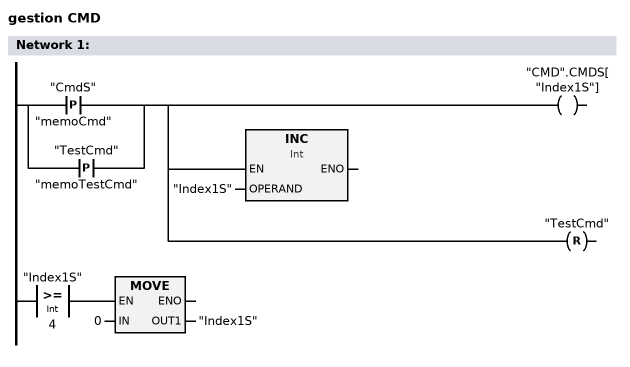
   RUNG wire#powerrail
      P_Contact(operand := "CmdS", bit := "memoCmd")
      wire#w1
      Coil( "CMD".CMDS["Index1S"] )
   END_RUNG
   RUNG wire#powerrail
      P_Contact(operand := "TestCmd", bit := "memoTestCmd")
   END_RUNG wire#w1
   RUNG wire#w1
      { S7_Templates := "DestType := Int" } Inc( "Index1S" )
   END_RUNG
   RUNG wire#w1
      R_Coil( "TestCmd" )
   END_RUNG
   RUNG wire#powerrail
      { S7_Templates := "SrcType := Int" } GE_Contact(in1 := "Index1S", in2 := 4)
      Move(in := 0, out1 => "Index1S")
   END_RUNG
   // the same network as SCL:
   #_w1 := "CmdS" AND NOT "memoCmd";   // rising edge of "CmdS"
   "memoCmd" := "CmdS";
   #_w2 := "TestCmd" AND NOT "memoTestCmd";   // rising edge of "TestCmd"
   "memoTestCmd" := "TestCmd";
   "CMD".CMDS["Index1S"] := #_w1 OR #_w2;
   IF #_w1 OR #_w2 THEN
       "Index1S" := "Index1S" + 1;
       "TestCmd" := FALSE;
   END_IF;
   IF "Index1S" >= 4 THEN "Index1S" := 0; END_IF;
END_REGION

REGION Network 2 (SCL)
   IF "TestX40" AND NOT "CMD".CMDFinal_S THEN
       IF "CMD".CMDS["index2S"] = TRUE THEN
           "CMD".CMDFinal_S := TRUE;
           "CMD".CMDS["index2S"] := 0;
       ELSE
           "index2S" := "index2S" + 1;
           IF "index2S" >= 4 THEN
               "index2S" := 0;
           END_IF;
       END_IF;
   END_IF;
END_REGION
END_FUNCTION

ORGANIZATION_BLOCK "Main"   // OB1, LAD, ProgramCycle
{ S7_Optimized_Access := 'TRUE' }
VERSION : 0.1
   VAR_INPUT
      Initial_Call : Bool;
      Remanence : Bool;
   END_VAR
BEGIN

REGION Network 1
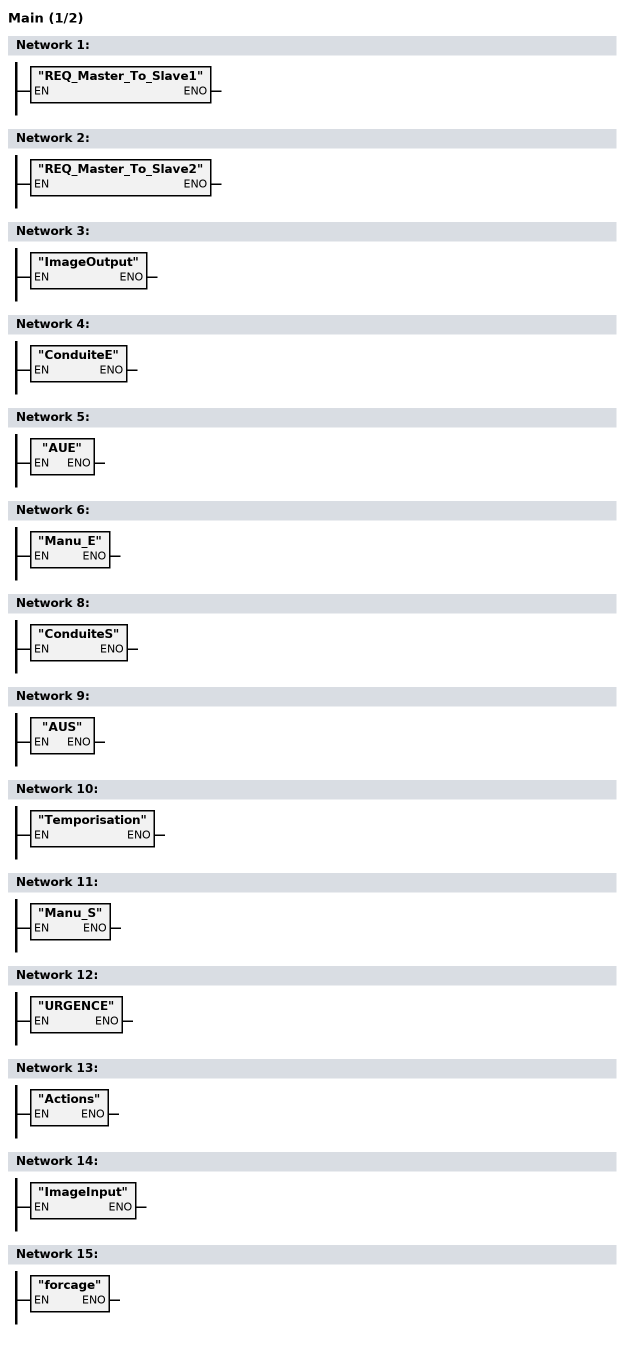
   RUNG wire#powerrail
      "REQ_Master_To_Slave1"()
   END_RUNG
   // the same network as SCL:
   "REQ_Master_To_Slave1"();
END_REGION

REGION Network 2
   RUNG wire#powerrail
      "REQ_Master_To_Slave2"()
   END_RUNG
   // the same network as SCL:
   "REQ_Master_To_Slave2"();
END_REGION

REGION Network 3
   RUNG wire#powerrail
      "ImageOutput"()
   END_RUNG
   // the same network as SCL:
   "ImageOutput"();
END_REGION

REGION Network 4
   RUNG wire#powerrail
      "ConduiteE"()
   END_RUNG
   // the same network as SCL:
   "ConduiteE"();
END_REGION

REGION Network 5
   RUNG wire#powerrail
      "AUE"()
   END_RUNG
   // the same network as SCL:
   "AUE"();
END_REGION

REGION Network 6
   RUNG wire#powerrail
      "Manu_E"()
   END_RUNG
   // the same network as SCL:
   "Manu_E"();
END_REGION

REGION Network 8
   RUNG wire#powerrail
      "ConduiteS"()
   END_RUNG
   // the same network as SCL:
   "ConduiteS"();
END_REGION

REGION Network 9
   RUNG wire#powerrail
      "AUS"()
   END_RUNG
   // the same network as SCL:
   "AUS"();
END_REGION

REGION Network 10
   RUNG wire#powerrail
      "Temporisation"()
   END_RUNG
   // the same network as SCL:
   "Temporisation"();
END_REGION

REGION Network 11
   RUNG wire#powerrail
      "Manu_S"()
   END_RUNG
   // the same network as SCL:
   "Manu_S"();
END_REGION

REGION Network 12
   RUNG wire#powerrail
      "URGENCE"()
   END_RUNG
   // the same network as SCL:
   "URGENCE"();
END_REGION

REGION Network 13
   RUNG wire#powerrail
      "Actions"()
   END_RUNG
   // the same network as SCL:
   "Actions"();
END_REGION

REGION Network 14
   RUNG wire#powerrail
      "ImageInput"()
   END_RUNG
   // the same network as SCL:
   "ImageInput"();
END_REGION

REGION Network 15
   RUNG wire#powerrail
      "forcage"()
   END_RUNG
   // the same network as SCL:
   "forcage"();
END_REGION

REGION Network 16
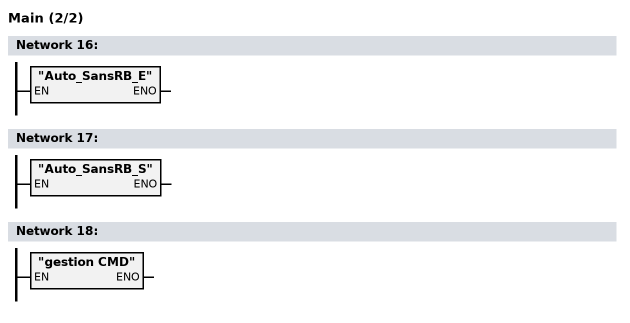
   RUNG wire#powerrail
      "Auto_SansRB_E"()
   END_RUNG
   // the same network as SCL:
   "Auto_SansRB_E"();
END_REGION

REGION Network 17
   RUNG wire#powerrail
      "Auto_SansRB_S"()
   END_RUNG
   // the same network as SCL:
   "Auto_SansRB_S"();
END_REGION

REGION Network 18
   RUNG wire#powerrail
      "gestion CMD"()
   END_RUNG
   // the same network as SCL:
   "gestion CMD"();
END_REGION
END_ORGANIZATION_BLOCK

ORGANIZATION_BLOCK "Startup"   // OB100, LAD, Startup
TITLE = "Complete Restart"
{ S7_Optimized_Access := 'TRUE' }
VERSION : 0.1
   VAR_INPUT
      LostRetentive : Bool;   // True if retentive data are lost
      LostRTC : Bool;   // True if date and time are lost
   END_VAR
BEGIN

REGION Network 1
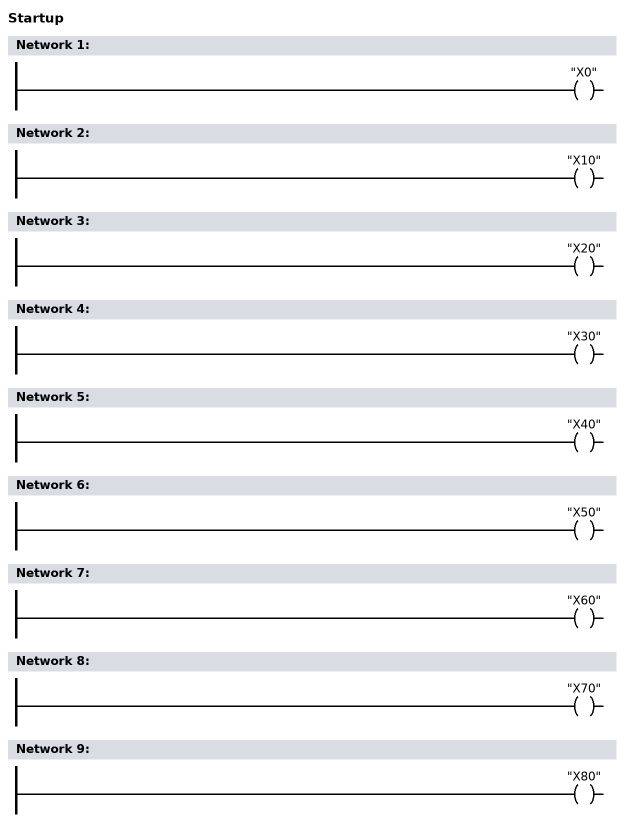
   RUNG wire#powerrail
      Coil( "X0" )
   END_RUNG
   // the same network as SCL:
   "X0" := TRUE;
END_REGION

REGION Network 2
   RUNG wire#powerrail
      Coil( "X10" )
   END_RUNG
   // the same network as SCL:
   "X10" := TRUE;
END_REGION

REGION Network 3
   RUNG wire#powerrail
      Coil( "X20" )
   END_RUNG
   // the same network as SCL:
   "X20" := TRUE;
END_REGION

REGION Network 4
   RUNG wire#powerrail
      Coil( "X30" )
   END_RUNG
   // the same network as SCL:
   "X30" := TRUE;
END_REGION

REGION Network 5
   RUNG wire#powerrail
      Coil( "X40" )
   END_RUNG
   // the same network as SCL:
   "X40" := TRUE;
END_REGION

REGION Network 6
   RUNG wire#powerrail
      Coil( "X50" )
   END_RUNG
   // the same network as SCL:
   "X50" := TRUE;
END_REGION

REGION Network 7
   RUNG wire#powerrail
      Coil( "X60" )
   END_RUNG
   // the same network as SCL:
   "X60" := TRUE;
END_REGION

REGION Network 8
   RUNG wire#powerrail
      Coil( "X70" )
   END_RUNG
   // the same network as SCL:
   "X70" := TRUE;
END_REGION

REGION Network 9
   RUNG wire#powerrail
      Coil( "X80" )
   END_RUNG
   // the same network as SCL:
   "X80" := TRUE;
END_REGION
END_ORGANIZATION_BLOCK